(*	| author		| Beckhoff Automation Poland	|	*)
(* 	-------------------------------------------------	*)
(*	| wersion		| 3.0							|	*)
(* 	-------------------------------------------------	*)
(*	| TC version	| 3.1.4024.7					| 	*)
(* 	-------------------------------------------------	*)
(*	| date			| 19.05.2020					|	*)
(* 	-------------------------------------------------	*)
(*	| description	| sample visu with navigation		
					  and frequently used functions	|  	*)
PROGRAM MAIN
VAR
END_VAR

P_HmiControl();
P_UserControl();
P_SystemInfo();
P_TaskInfo();
P_PersistentData();
P_Events();
P_FileDialog();
P_Table();
P_ControllerInfo();
P_CloseTcHmiExe();

END_PROGRAM

(* stored: Version 1.1.0.1, ProductVersion 3.1.4024.3
   POU MAIN: Id {4827b60d-9066-4abc-9b71-8a8a14f3e433}, SpecialFunc None *)
